FUNCTION_BLOCK FB_String
VAR_INPUT
    sInput : STRING;
END_VAR
VAR_OUTPUT
    sOutput : STRING;
END_VAR

sOutput := CONCAT('Value: ', sInput);

END_FUNCTION_BLOCK

(* stored: Version 1.1.0.1, ProductVersion 3.1.4024.10
   POU FB_String: KindOfPOU Element *)
